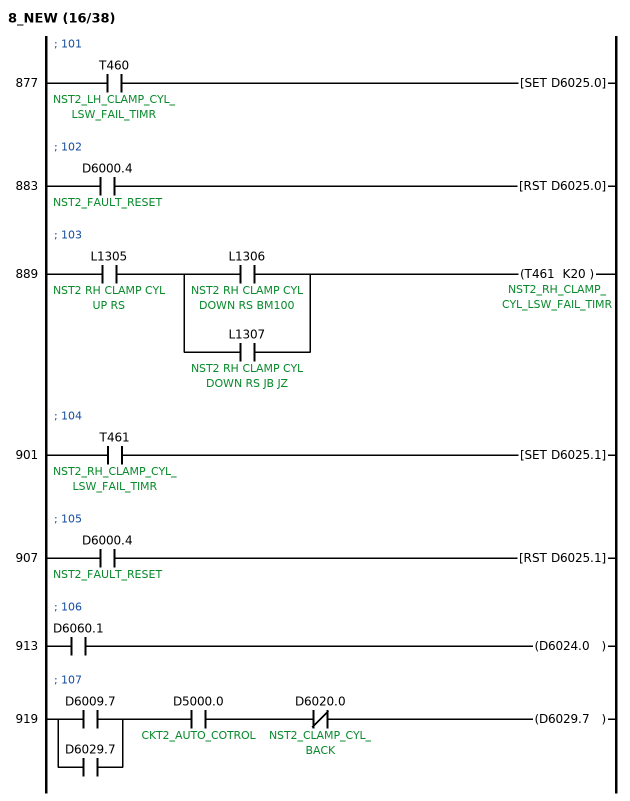
[picture p96: ladder of 8_NEW, rungs at steps 877 to 919]
; 101
877   LD      T460  ; NST2_LH_CLAMP_CYL_LSW_FAIL_TIMR
      SET     D6025.0
; 102
883   LD      D6000.4  ; NST2_FAULT_RESET
      RST     D6025.0
; 103
889   LD      L1305  ; NST2 RH CLAMP CYL UP RS
      LD      L1306  ; NST2 RH CLAMP CYL DOWN RS BM100
      OR      L1307  ; NST2 RH CLAMP CYL DOWN RS JB JZ
      ANB
      OUT     T461 K20  ; NST2_RH_CLAMP_CYL_LSW_FAIL_TIMR
; 104
901   LD      T461  ; NST2_RH_CLAMP_CYL_LSW_FAIL_TIMR
      SET     D6025.1
; 105
907   LD      D6000.4  ; NST2_FAULT_RESET
      RST     D6025.1
; 106
913   LD      D6060.1
      OUT     D6024.0
; 107
919   LD      D6009.7
      OR      D6029.7
      AND     D5000.0  ; CKT2_AUTO_COTROL
      ANI     D6020.0  ; NST2_CLAMP_CYL_BACK
      OUT     D6029.7
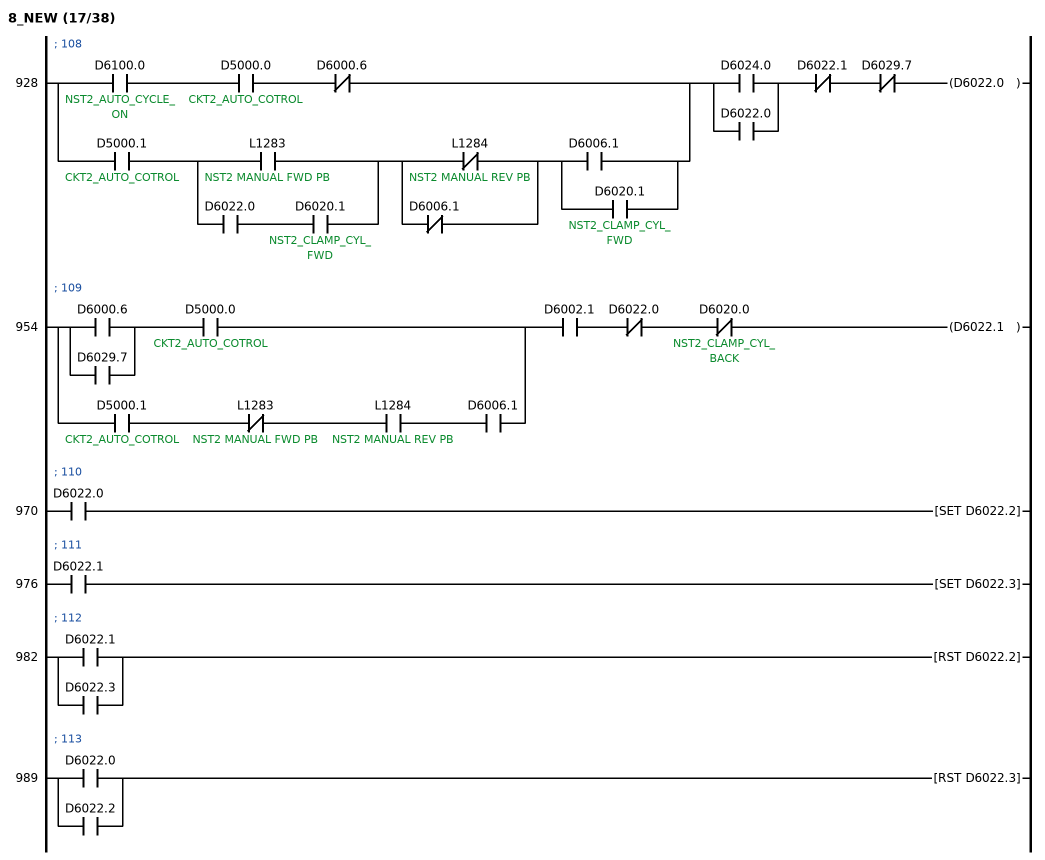
; 108
928   LD      D6100.0  ; NST2_AUTO_CYCLE_ON
      AND     D5000.0  ; CKT2_AUTO_COTROL
      ANI     D6000.6
      LD      D5000.1  ; CKT2_AUTO_COTROL
      LD      L1283  ; NST2 MANUAL FWD PB
      LD      D6022.0
      AND     D6020.1  ; NST2_CLAMP_CYL_FWD
      ORB
      ANB
      LDI     L1284  ; NST2 MANUAL REV PB
      ORI     D6006.1
      ANB
      LD      D6006.1
      OR      D6020.1  ; NST2_CLAMP_CYL_FWD
      ANB
      ORB
      LD      D6024.0
      OR      D6022.0
      ANB
      ANI     D6022.1
      ANI     D6029.7
      OUT     D6022.0
; 109
954   LD      D6000.6
      OR      D6029.7
      AND     D5000.0  ; CKT2_AUTO_COTROL
      LD      D5000.1  ; CKT2_AUTO_COTROL
      ANI     L1283  ; NST2 MANUAL FWD PB
      AND     L1284  ; NST2 MANUAL REV PB
      AND     D6006.1
      ORB
      AND     D6002.1
      ANI     D6022.0
      ANI     D6020.0  ; NST2_CLAMP_CYL_BACK
      OUT     D6022.1
; 110
970   LD      D6022.0
      SET     D6022.2
; 111
976   LD      D6022.1
      SET     D6022.3
; 112
982   LD      D6022.1
      OR      D6022.3
      RST     D6022.2
; 113
989   LD      D6022.0
      OR      D6022.2
      RST     D6022.3
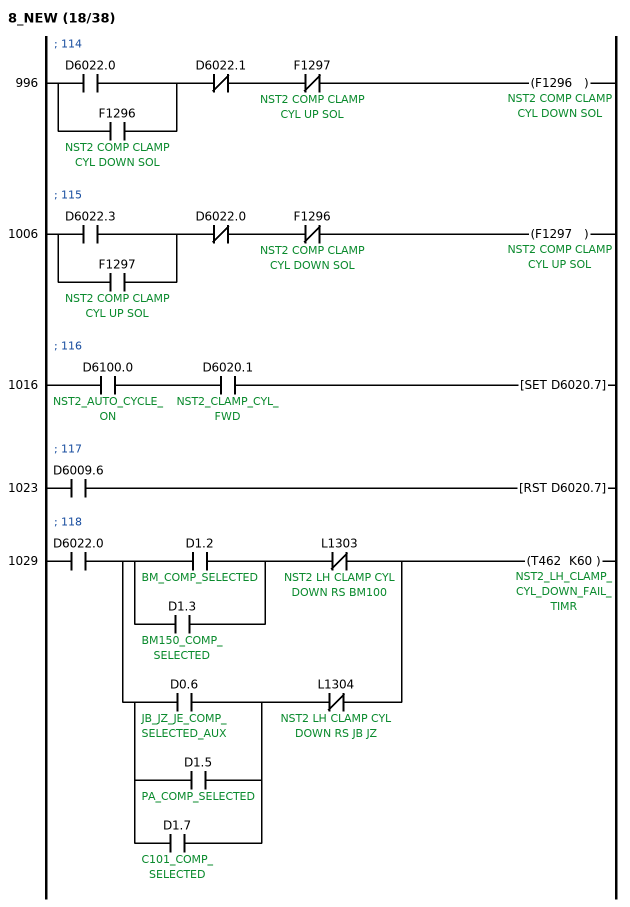
; 114
996   LD      D6022.0
      OR      F1296  ; NST2 COMP CLAMP CYL DOWN SOL
      ANI     D6022.1
      ANI     F1297  ; NST2 COMP CLAMP CYL UP SOL
      OUT     F1296  ; NST2 COMP CLAMP CYL DOWN SOL
; 115
1006  LD      D6022.3
      OR      F1297  ; NST2 COMP CLAMP CYL UP SOL
      ANI     D6022.0
      ANI     F1296  ; NST2 COMP CLAMP CYL DOWN SOL
      OUT     F1297  ; NST2 COMP CLAMP CYL UP SOL
; 116
1016  LD      D6100.0  ; NST2_AUTO_CYCLE_ON
      AND     D6020.1  ; NST2_CLAMP_CYL_FWD
      SET     D6020.7
; 117
1023  LD      D6009.6
      RST     D6020.7
; 118
1029  LD      D6022.0
      LD      D1.2  ; BM_COMP_SELECTED
      OR      D1.3  ; BM150_COMP_SELECTED
      ANI     L1303  ; NST2 LH CLAMP CYL DOWN RS BM100
      LD      D0.6  ; JB_JZ_JE_COMP_SELECTED_AUX
      OR      D1.5  ; PA_COMP_SELECTED
      OR      D1.7  ; C101_COMP_SELECTED
      ANI     L1304  ; NST2 LH CLAMP CYL DOWN RS JB JZ
      ORB
      ANB
      OUT     T462 K60  ; NST2_LH_CLAMP_CYL_DOWN_FAIL_TIMR
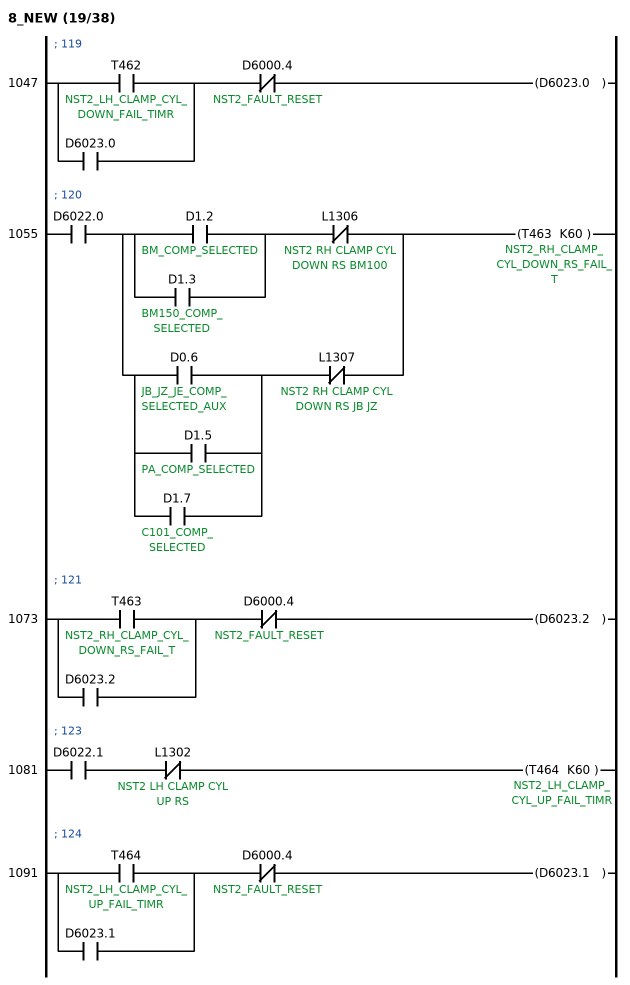
; 119
1047  LD      T462  ; NST2_LH_CLAMP_CYL_DOWN_FAIL_TIMR
      OR      D6023.0
      ANI     D6000.4  ; NST2_FAULT_RESET
      OUT     D6023.0
; 120
1055  LD      D6022.0
      LD      D1.2  ; BM_COMP_SELECTED
      OR      D1.3  ; BM150_COMP_SELECTED
      ANI     L1306  ; NST2 RH CLAMP CYL DOWN RS BM100
      LD      D0.6  ; JB_JZ_JE_COMP_SELECTED_AUX
      OR      D1.5  ; PA_COMP_SELECTED
      OR      D1.7  ; C101_COMP_SELECTED
      ANI     L1307  ; NST2 RH CLAMP CYL DOWN RS JB JZ
      ORB
      ANB
      OUT     T463 K60  ; NST2_RH_CLAMP_CYL_DOWN_RS_FAIL_T
; 121
1073  LD      T463  ; NST2_RH_CLAMP_CYL_DOWN_RS_FAIL_T
      OR      D6023.2
      ANI     D6000.4  ; NST2_FAULT_RESET
      OUT     D6023.2
; 123
1081  LD      D6022.1
      ANI     L1302  ; NST2 LH CLAMP CYL UP RS
      OUT     T464 K60  ; NST2_LH_CLAMP_CYL_UP_FAIL_TIMR
; 124
1091  LD      T464  ; NST2_LH_CLAMP_CYL_UP_FAIL_TIMR
      OR      D6023.1
      ANI     D6000.4  ; NST2_FAULT_RESET
      OUT     D6023.1
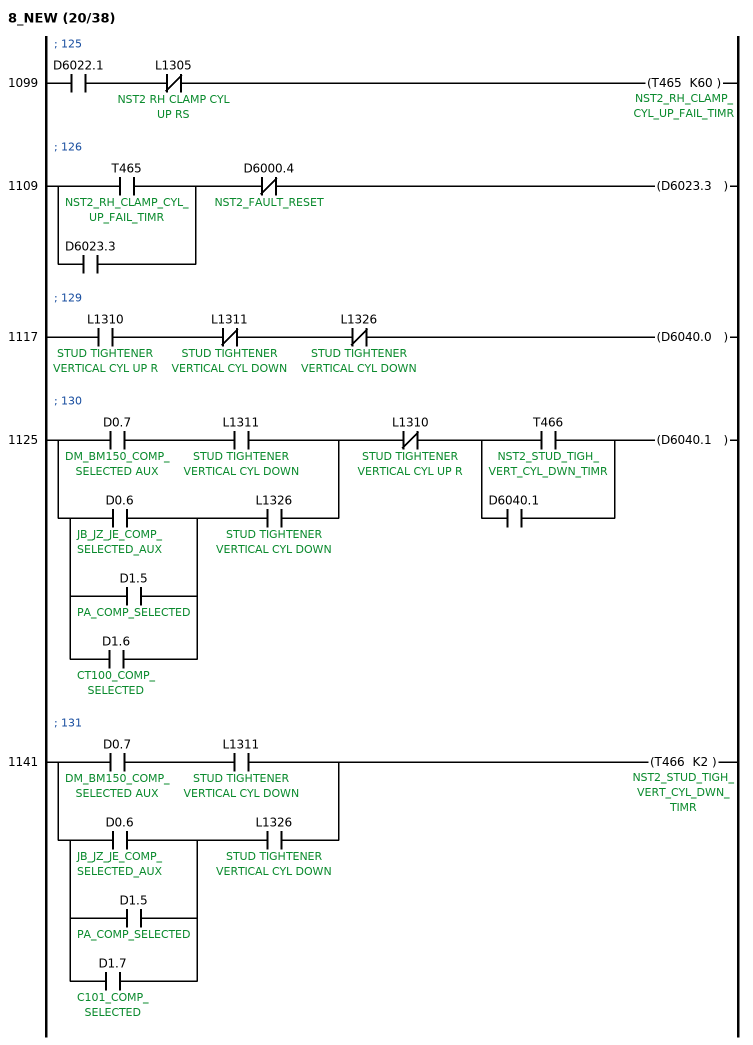
; 125
1099  LD      D6022.1
      ANI     L1305  ; NST2 RH CLAMP CYL UP RS
      OUT     T465 K60  ; NST2_RH_CLAMP_CYL_UP_FAIL_TIMR
; 126
1109  LD      T465  ; NST2_RH_CLAMP_CYL_UP_FAIL_TIMR
      OR      D6023.3
      ANI     D6000.4  ; NST2_FAULT_RESET
      OUT     D6023.3
; 129
1117  LD      L1310  ; STUD TIGHTENER VERTICAL CYL UP R
      ANI     L1311  ; STUD TIGHTENER VERTICAL CYL DOWN
      ANI     L1326  ; STUD TIGHTENER VERTICAL CYL DOWN
      OUT     D6040.0
; 130
1125  LD      D0.7  ; DM_BM150_COMP_SELECTED AUX
      AND     L1311  ; STUD TIGHTENER VERTICAL CYL DOWN
      LD      D0.6  ; JB_JZ_JE_COMP_SELECTED_AUX
      OR      D1.5  ; PA_COMP_SELECTED
      OR      D1.6  ; CT100_COMP_SELECTED
      AND     L1326  ; STUD TIGHTENER VERTICAL CYL DOWN
      ORB
      ANI     L1310  ; STUD TIGHTENER VERTICAL CYL UP R
      LD      T466  ; NST2_STUD_TIGH_VERT_CYL_DWN_TIMR
      OR      D6040.1
      ANB
      OUT     D6040.1
; 131
1141  LD      D0.7  ; DM_BM150_COMP_SELECTED AUX
      AND     L1311  ; STUD TIGHTENER VERTICAL CYL DOWN
      LD      D0.6  ; JB_JZ_JE_COMP_SELECTED_AUX
      OR      D1.5  ; PA_COMP_SELECTED
      OR      D1.7  ; C101_COMP_SELECTED
      AND     L1326  ; STUD TIGHTENER VERTICAL CYL DOWN
      ORB
      OUT     T466 K2  ; NST2_STUD_TIGH_VERT_CYL_DWN_TIMR
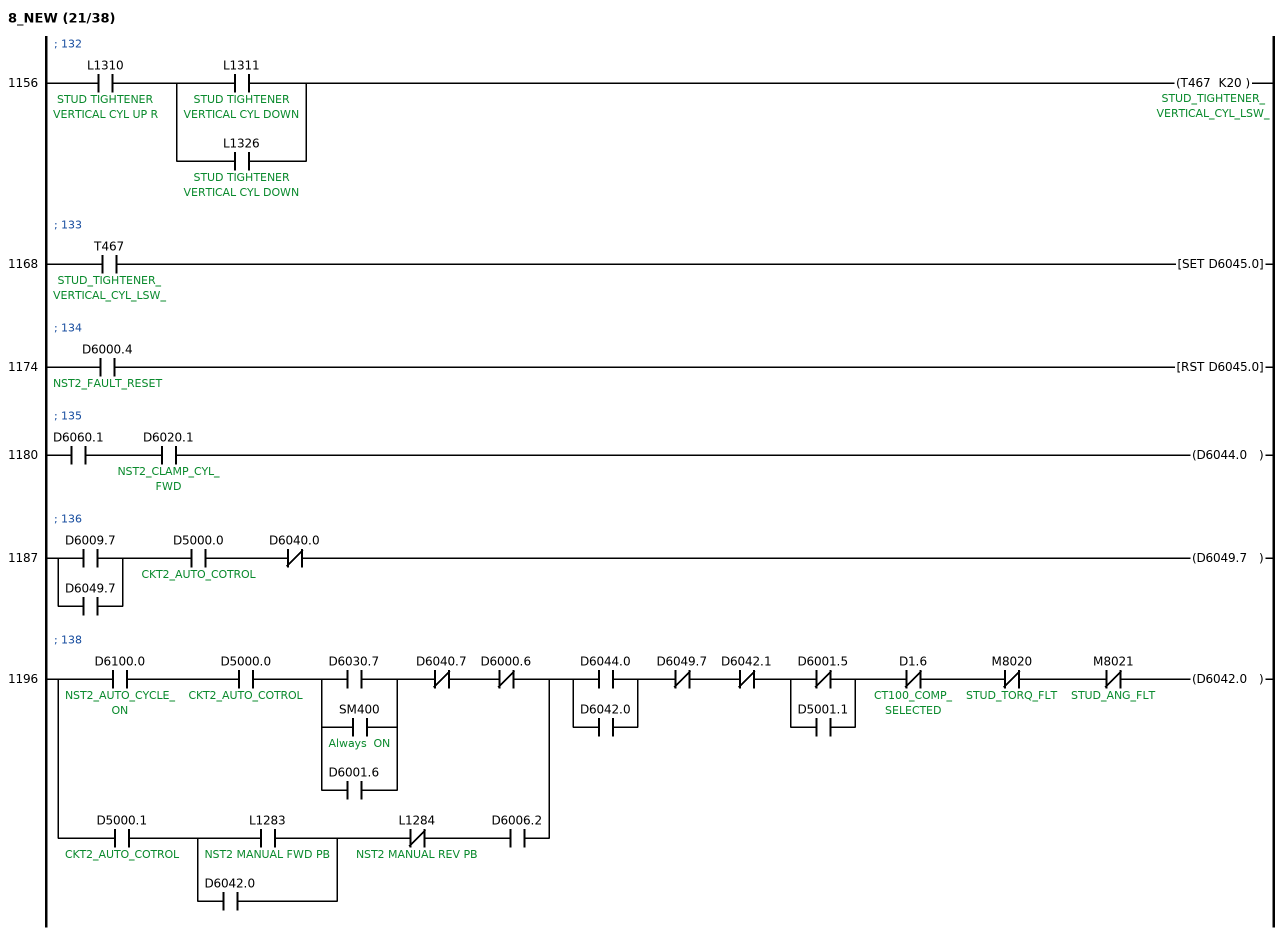
; 132
1156  LD      L1310  ; STUD TIGHTENER VERTICAL CYL UP R
      LD      L1311  ; STUD TIGHTENER VERTICAL CYL DOWN
      OR      L1326  ; STUD TIGHTENER VERTICAL CYL DOWN
      ANB
      OUT     T467 K20  ; STUD_TIGHTENER_VERTICAL_CYL_LSW_
; 133
1168  LD      T467  ; STUD_TIGHTENER_VERTICAL_CYL_LSW_
      SET     D6045.0
; 134
1174  LD      D6000.4  ; NST2_FAULT_RESET
      RST     D6045.0
; 135
1180  LD      D6060.1
      AND     D6020.1  ; NST2_CLAMP_CYL_FWD
      OUT     D6044.0
; 136
1187  LD      D6009.7
      OR      D6049.7
      AND     D5000.0  ; CKT2_AUTO_COTROL
      ANI     D6040.0
      OUT     D6049.7
; 138
1196  LD      D6100.0  ; NST2_AUTO_CYCLE_ON
      AND     D5000.0  ; CKT2_AUTO_COTROL
      LD      D6030.7
      OR      SM400  ; Always  ON
      OR      D6001.6
      ANB
      ANI     D6040.7
      ANI     D6000.6
      LD      D5000.1  ; CKT2_AUTO_COTROL
      LD      L1283  ; NST2 MANUAL FWD PB
      OR      D6042.0
      ANB
      ANI     L1284  ; NST2 MANUAL REV PB
      AND     D6006.2
      ORB
      LD      D6044.0
      OR      D6042.0
      ANB
      ANI     D6049.7
      ANI     D6042.1
      LDI     D6001.5
      OR      D5001.1
      ANB
      ANI     D1.6  ; CT100_COMP_SELECTED
      ANI     M8020  ; STUD_TORQ_FLT
      ANI     M8021  ; STUD_ANG_FLT
      OUT     D6042.0
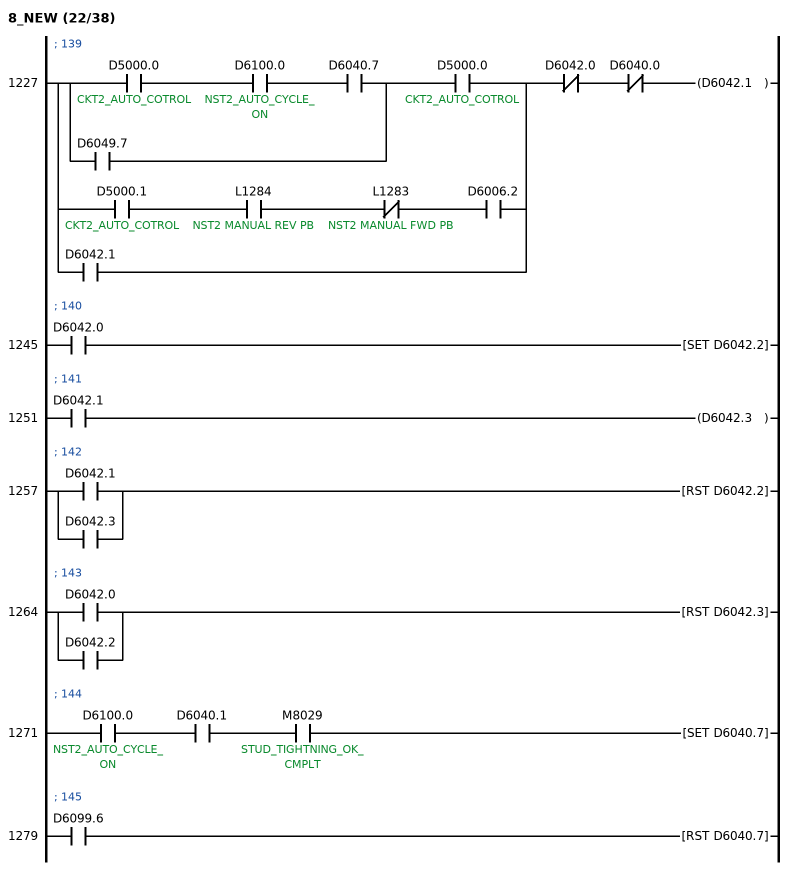
; 139
1227  LD      D5000.0  ; CKT2_AUTO_COTROL
      AND     D6100.0  ; NST2_AUTO_CYCLE_ON
      AND     D6040.7
      OR      D6049.7
      AND     D5000.0  ; CKT2_AUTO_COTROL
      LD      D5000.1  ; CKT2_AUTO_COTROL
      AND     L1284  ; NST2 MANUAL REV PB
      ANI     L1283  ; NST2 MANUAL FWD PB
      AND     D6006.2
      ORB
      OR      D6042.1
      ANI     D6042.0
      ANI     D6040.0
      OUT     D6042.1
; 140
1245  LD      D6042.0
      SET     D6042.2
; 141
1251  LD      D6042.1
      OUT     D6042.3
; 142
1257  LD      D6042.1
      OR      D6042.3
      RST     D6042.2
; 143
1264  LD      D6042.0
      OR      D6042.2
      RST     D6042.3
; 144
1271  LD      D6100.0  ; NST2_AUTO_CYCLE_ON
      AND     D6040.1
      AND     M8029  ; STUD_TIGHTNING_OK_CMPLT
      SET     D6040.7
; 145
1279  LD      D6099.6
      RST     D6040.7
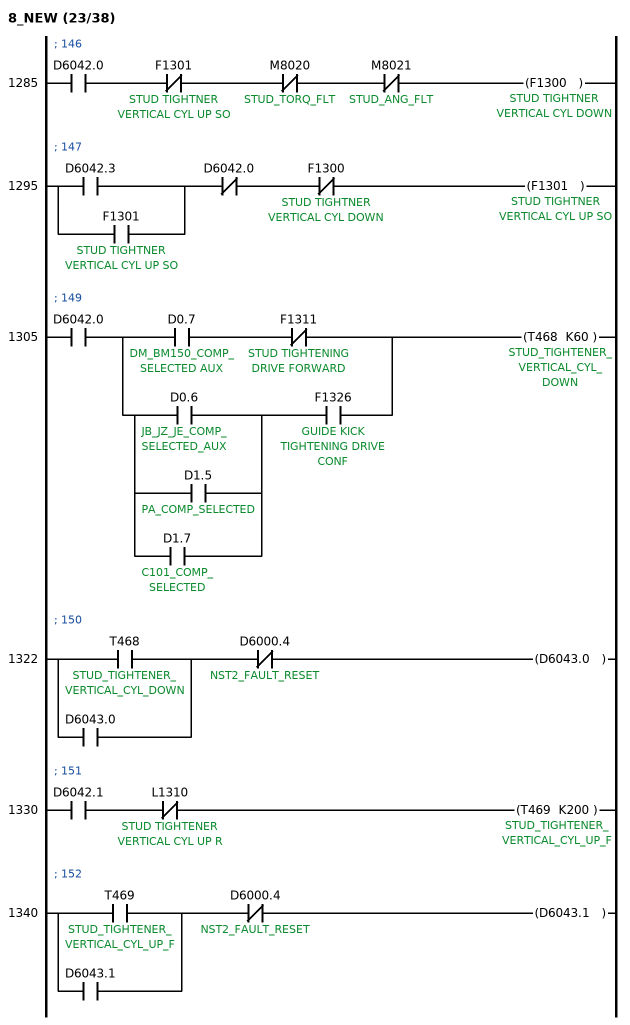
; 146
1285  LD      D6042.0
      ANI     F1301  ; STUD TIGHTNER VERTICAL CYL UP SO
      ANI     M8020  ; STUD_TORQ_FLT
      ANI     M8021  ; STUD_ANG_FLT
      OUT     F1300  ; STUD TIGHTNER VERTICAL CYL DOWN
; 147
1295  LD      D6042.3
      OR      F1301  ; STUD TIGHTNER VERTICAL CYL UP SO
      ANI     D6042.0
      ANI     F1300  ; STUD TIGHTNER VERTICAL CYL DOWN
      OUT     F1301  ; STUD TIGHTNER VERTICAL CYL UP SO
; 149
1305  LD      D6042.0
      LD      D0.7  ; DM_BM150_COMP_SELECTED AUX
      ANI     F1311  ; STUD TIGHTENING DRIVE FORWARD
      LD      D0.6  ; JB_JZ_JE_COMP_SELECTED_AUX
      OR      D1.5  ; PA_COMP_SELECTED
      OR      D1.7  ; C101_COMP_SELECTED
      AND     F1326  ; GUIDE KICK TIGHTENING DRIVE CONF
      ORB
      ANB
      OUT     T468 K60  ; STUD_TIGHTENER_VERTICAL_CYL_DOWN
; 150
1322  LD      T468  ; STUD_TIGHTENER_VERTICAL_CYL_DOWN
      OR      D6043.0
      ANI     D6000.4  ; NST2_FAULT_RESET
      OUT     D6043.0
; 151
1330  LD      D6042.1
      ANI     L1310  ; STUD TIGHTENER VERTICAL CYL UP R
      OUT     T469 K200  ; STUD_TIGHTENER_VERTICAL_CYL_UP_F
; 152
1340  LD      T469  ; STUD_TIGHTENER_VERTICAL_CYL_UP_F
      OR      D6043.1
      ANI     D6000.4  ; NST2_FAULT_RESET
      OUT     D6043.1
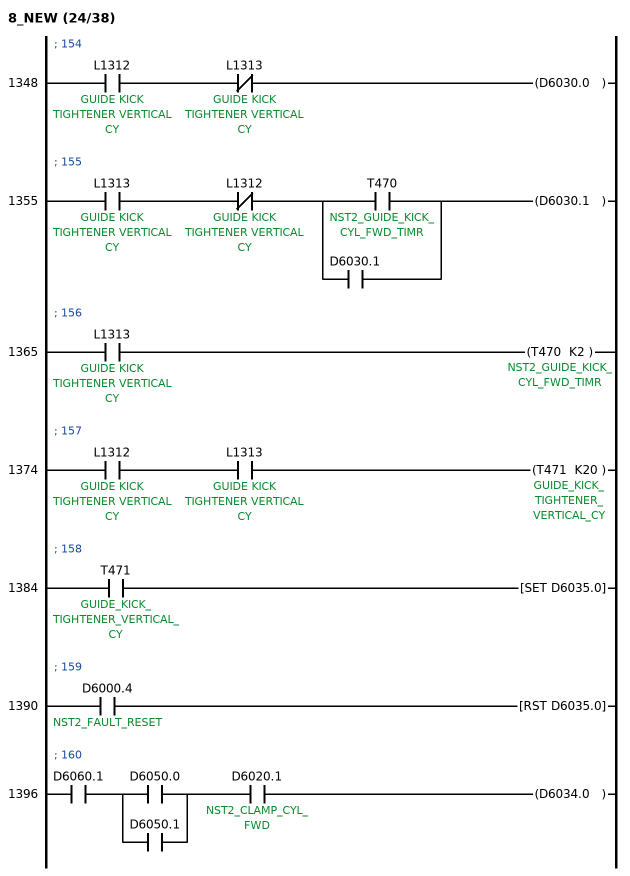
; 154
1348  LD      L1312  ; GUIDE KICK TIGHTENER VERTICAL CY
      ANI     L1313  ; GUIDE KICK TIGHTENER VERTICAL CY
      OUT     D6030.0
; 155
1355  LD      L1313  ; GUIDE KICK TIGHTENER VERTICAL CY
      ANI     L1312  ; GUIDE KICK TIGHTENER VERTICAL CY
      LD      T470  ; NST2_GUIDE_KICK_CYL_FWD_TIMR
      OR      D6030.1
      ANB
      OUT     D6030.1
; 156
1365  LD      L1313  ; GUIDE KICK TIGHTENER VERTICAL CY
      OUT     T470 K2  ; NST2_GUIDE_KICK_CYL_FWD_TIMR
; 157
1374  LD      L1312  ; GUIDE KICK TIGHTENER VERTICAL CY
      AND     L1313  ; GUIDE KICK TIGHTENER VERTICAL CY
      OUT     T471 K20  ; GUIDE_KICK_TIGHTENER_VERTICAL_CY
; 158
1384  LD      T471  ; GUIDE_KICK_TIGHTENER_VERTICAL_CY
      SET     D6035.0
; 159
1390  LD      D6000.4  ; NST2_FAULT_RESET
      RST     D6035.0
; 160
1396  LD      D6060.1
      LD      D6050.0
      OR      D6050.1
      ANB
      AND     D6020.1  ; NST2_CLAMP_CYL_FWD
      OUT     D6034.0
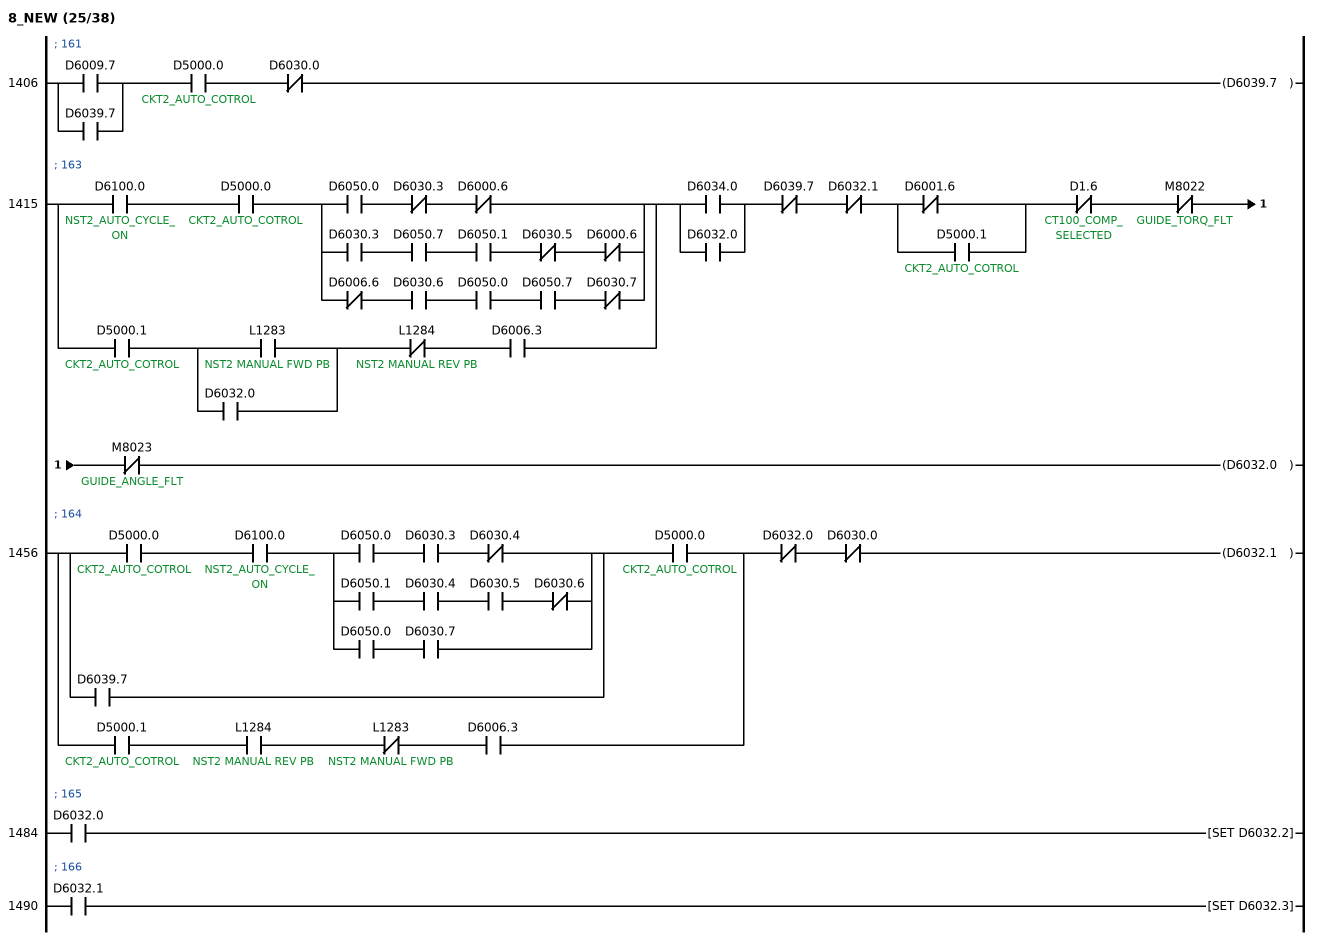
; 161
1406  LD      D6009.7
      OR      D6039.7
      AND     D5000.0  ; CKT2_AUTO_COTROL
      ANI     D6030.0
      OUT     D6039.7
; 163
1415  LD      D6100.0  ; NST2_AUTO_CYCLE_ON
      AND     D5000.0  ; CKT2_AUTO_COTROL
      LD      D6050.0
      ANI     D6030.3
      ANI     D6000.6
      LD      D6030.3
      AND     D6050.7
      AND     D6050.1
      ANI     D6030.5
      ANI     D6000.6
      ORB
      LDI     D6006.6
      AND     D6030.6
      AND     D6050.0
      AND     D6050.7
      ANI     D6030.7
      ORB
      ANB
      LD      D5000.1  ; CKT2_AUTO_COTROL
      LD      L1283  ; NST2 MANUAL FWD PB
      OR      D6032.0
      ANB
      ANI     L1284  ; NST2 MANUAL REV PB
      AND     D6006.3
      ORB
      LD      D6034.0
      OR      D6032.0
      ANB
      ANI     D6039.7
      ANI     D6032.1
      LDI     D6001.6
      OR      D5000.1  ; CKT2_AUTO_COTROL
      ANB
      ANI     D1.6  ; CT100_COMP_SELECTED
      ANI     M8022  ; GUIDE_TORQ_FLT
      ANI     M8023  ; GUIDE_ANGLE_FLT
      OUT     D6032.0
; 164
1456  LD      D5000.0  ; CKT2_AUTO_COTROL
      AND     D6100.0  ; NST2_AUTO_CYCLE_ON
      LD      D6050.0
      AND     D6030.3
      ANI     D6030.4
      LD      D6050.1
      AND     D6030.4
      AND     D6030.5
      ANI     D6030.6
      ORB
      LD      D6050.0
      AND     D6030.7
      ORB
      ANB
      OR      D6039.7
      AND     D5000.0  ; CKT2_AUTO_COTROL
      LD      D5000.1  ; CKT2_AUTO_COTROL
      AND     L1284  ; NST2 MANUAL REV PB
      ANI     L1283  ; NST2 MANUAL FWD PB
      AND     D6006.3
      ORB
      ANI     D6032.0
      ANI     D6030.0
      OUT     D6032.1
; 165
1484  LD      D6032.0
      SET     D6032.2
; 166
1490  LD      D6032.1
      SET     D6032.3
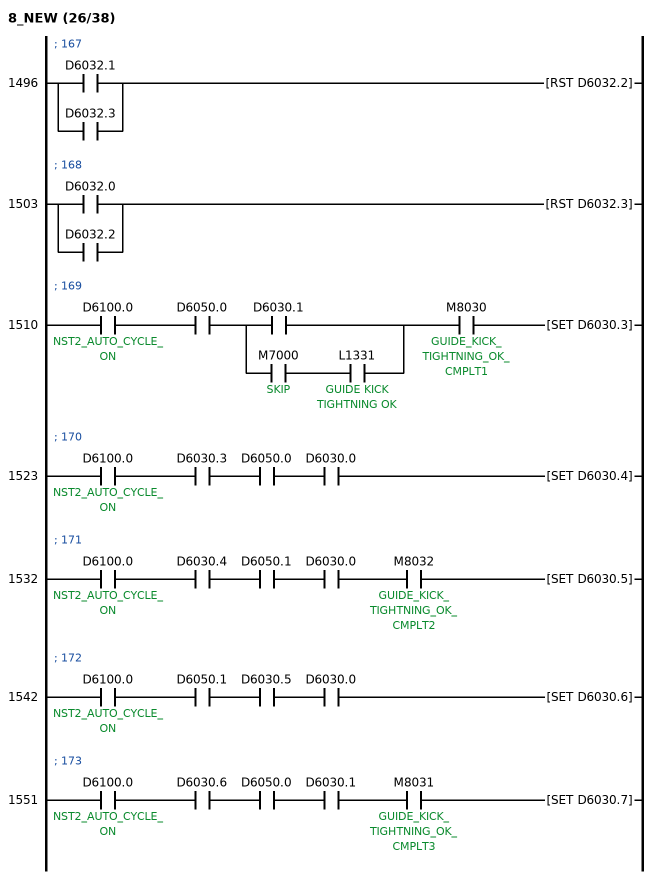
; 167
1496  LD      D6032.1
      OR      D6032.3
      RST     D6032.2
; 168
1503  LD      D6032.0
      OR      D6032.2
      RST     D6032.3
; 169
1510  LD      D6100.0  ; NST2_AUTO_CYCLE_ON
      AND     D6050.0
      LD      D6030.1
      LD      M7000  ; SKIP
      AND     L1331  ; GUIDE KICK TIGHTNING OK
      ORB
      ANB
      AND     M8030  ; GUIDE_KICK_TIGHTNING_OK_CMPLT1
      SET     D6030.3
; 170
1523  LD      D6100.0  ; NST2_AUTO_CYCLE_ON
      AND     D6030.3
      AND     D6050.0
      AND     D6030.0
      SET     D6030.4
; 171
1532  LD      D6100.0  ; NST2_AUTO_CYCLE_ON
      AND     D6030.4
      AND     D6050.1
      AND     D6030.0
      AND     M8032  ; GUIDE_KICK_TIGHTNING_OK_CMPLT2
      SET     D6030.5
; 172
1542  LD      D6100.0  ; NST2_AUTO_CYCLE_ON
      AND     D6050.1
      AND     D6030.5
      AND     D6030.0
      SET     D6030.6
; 173
1551  LD      D6100.0  ; NST2_AUTO_CYCLE_ON
      AND     D6030.6
      AND     D6050.0
      AND     D6030.1
      AND     M8031  ; GUIDE_KICK_TIGHTNING_OK_CMPLT3
      SET     D6030.7
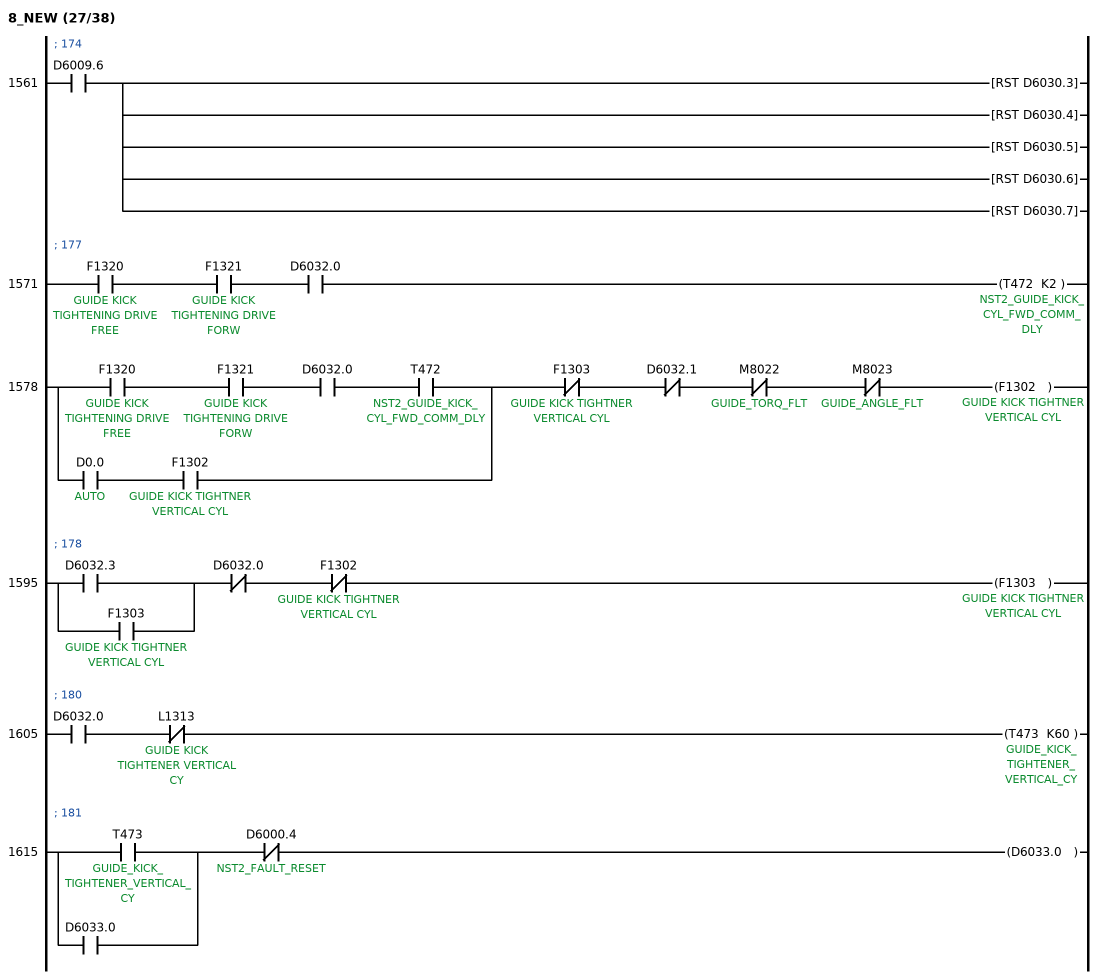
; 174
1561  LD      D6009.6
      RST     D6030.3
      RST     D6030.4
      RST     D6030.5
      RST     D6030.6
      RST     D6030.7
; 177
1571  LD      F1320  ; GUIDE KICK TIGHTENING DRIVE FREE
      AND     F1321  ; GUIDE KICK TIGHTENING DRIVE FORW
      AND     D6032.0
      OUT     T472 K2  ; NST2_GUIDE_KICK_CYL_FWD_COMM_DLY
1578  LD      F1320  ; GUIDE KICK TIGHTENING DRIVE FREE
      AND     F1321  ; GUIDE KICK TIGHTENING DRIVE FORW
      AND     D6032.0
      AND     T472  ; NST2_GUIDE_KICK_CYL_FWD_COMM_DLY
      LD      D0.0  ; AUTO
      AND     F1302  ; GUIDE KICK TIGHTNER VERTICAL CYL
      ORB
      ANI     F1303  ; GUIDE KICK TIGHTNER VERTICAL CYL
      ANI     D6032.1
      ANI     M8022  ; GUIDE_TORQ_FLT
      ANI     M8023  ; GUIDE_ANGLE_FLT
      OUT     F1302  ; GUIDE KICK TIGHTNER VERTICAL CYL
; 178
1595  LD      D6032.3
      OR      F1303  ; GUIDE KICK TIGHTNER VERTICAL CYL
      ANI     D6032.0
      ANI     F1302  ; GUIDE KICK TIGHTNER VERTICAL CYL
      OUT     F1303  ; GUIDE KICK TIGHTNER VERTICAL CYL
; 180
1605  LD      D6032.0
      ANI     L1313  ; GUIDE KICK TIGHTENER VERTICAL CY
      OUT     T473 K60  ; GUIDE_KICK_TIGHTENER_VERTICAL_CY
; 181
1615  LD      T473  ; GUIDE_KICK_TIGHTENER_VERTICAL_CY
      OR      D6033.0
      ANI     D6000.4  ; NST2_FAULT_RESET
      OUT     D6033.0
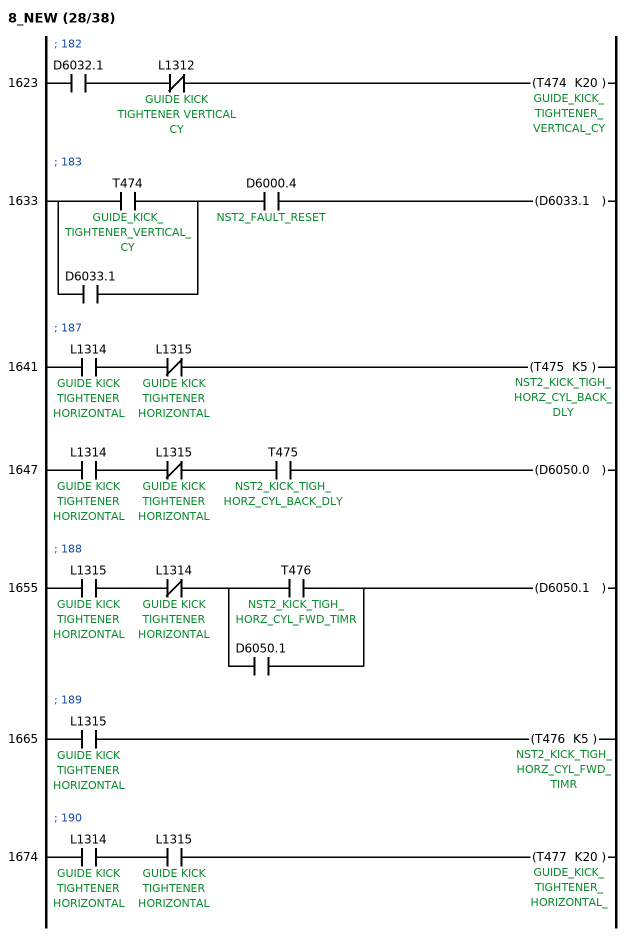
; 182
1623  LD      D6032.1
      ANI     L1312  ; GUIDE KICK TIGHTENER VERTICAL CY
      OUT     T474 K20  ; GUIDE_KICK_TIGHTENER_VERTICAL_CY
; 183
1633  LD      T474  ; GUIDE_KICK_TIGHTENER_VERTICAL_CY
      OR      D6033.1
      AND     D6000.4  ; NST2_FAULT_RESET
      OUT     D6033.1
; 187
1641  LD      L1314  ; GUIDE KICK TIGHTENER HORIZONTAL
      ANI     L1315  ; GUIDE KICK TIGHTENER HORIZONTAL
      OUT     T475 K5  ; NST2_KICK_TIGH_HORZ_CYL_BACK_DLY
1647  LD      L1314  ; GUIDE KICK TIGHTENER HORIZONTAL
      ANI     L1315  ; GUIDE KICK TIGHTENER HORIZONTAL
      AND     T475  ; NST2_KICK_TIGH_HORZ_CYL_BACK_DLY
      OUT     D6050.0
; 188
1655  LD      L1315  ; GUIDE KICK TIGHTENER HORIZONTAL
      ANI     L1314  ; GUIDE KICK TIGHTENER HORIZONTAL
      LD      T476  ; NST2_KICK_TIGH_HORZ_CYL_FWD_TIMR
      OR      D6050.1
      ANB
      OUT     D6050.1
; 189
1665  LD      L1315  ; GUIDE KICK TIGHTENER HORIZONTAL
      OUT     T476 K5  ; NST2_KICK_TIGH_HORZ_CYL_FWD_TIMR
; 190
1674  LD      L1314  ; GUIDE KICK TIGHTENER HORIZONTAL
      AND     L1315  ; GUIDE KICK TIGHTENER HORIZONTAL
      OUT     T477 K20  ; GUIDE_KICK_TIGHTENER_HORIZONTAL_
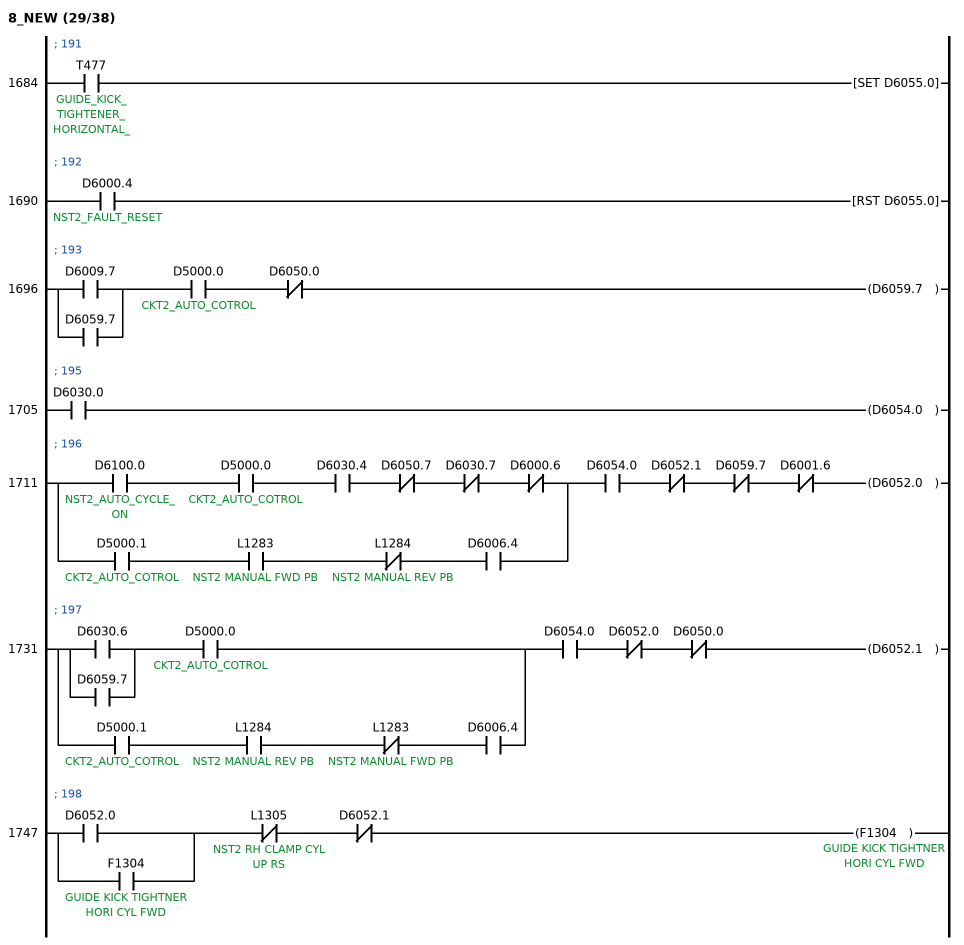
; 191
1684  LD      T477  ; GUIDE_KICK_TIGHTENER_HORIZONTAL_
      SET     D6055.0
; 192
1690  LD      D6000.4  ; NST2_FAULT_RESET
      RST     D6055.0
; 193
1696  LD      D6009.7
      OR      D6059.7
      AND     D5000.0  ; CKT2_AUTO_COTROL
      ANI     D6050.0
      OUT     D6059.7
; 195
1705  LD      D6030.0
      OUT     D6054.0
; 196
1711  LD      D6100.0  ; NST2_AUTO_CYCLE_ON
      AND     D5000.0  ; CKT2_AUTO_COTROL
      AND     D6030.4
      ANI     D6050.7
      ANI     D6030.7
      ANI     D6000.6
      LD      D5000.1  ; CKT2_AUTO_COTROL
      AND     L1283  ; NST2 MANUAL FWD PB
      ANI     L1284  ; NST2 MANUAL REV PB
      AND     D6006.4
      ORB
      AND     D6054.0
      ANI     D6052.1
      ANI     D6059.7
      ANI     D6001.6
      OUT     D6052.0
; 197
1731  LD      D6030.6
      OR      D6059.7
      AND     D5000.0  ; CKT2_AUTO_COTROL
      LD      D5000.1  ; CKT2_AUTO_COTROL
      AND     L1284  ; NST2 MANUAL REV PB
      ANI     L1283  ; NST2 MANUAL FWD PB
      AND     D6006.4
      ORB
      AND     D6054.0
      ANI     D6052.0
      ANI     D6050.0
      OUT     D6052.1
; 198
1747  LD      D6052.0
      OR      F1304  ; GUIDE KICK TIGHTNER HORI CYL FWD
      ANI     L1305  ; NST2 RH CLAMP CYL UP RS
      ANI     D6052.1
      OUT     F1304  ; GUIDE KICK TIGHTNER HORI CYL FWD
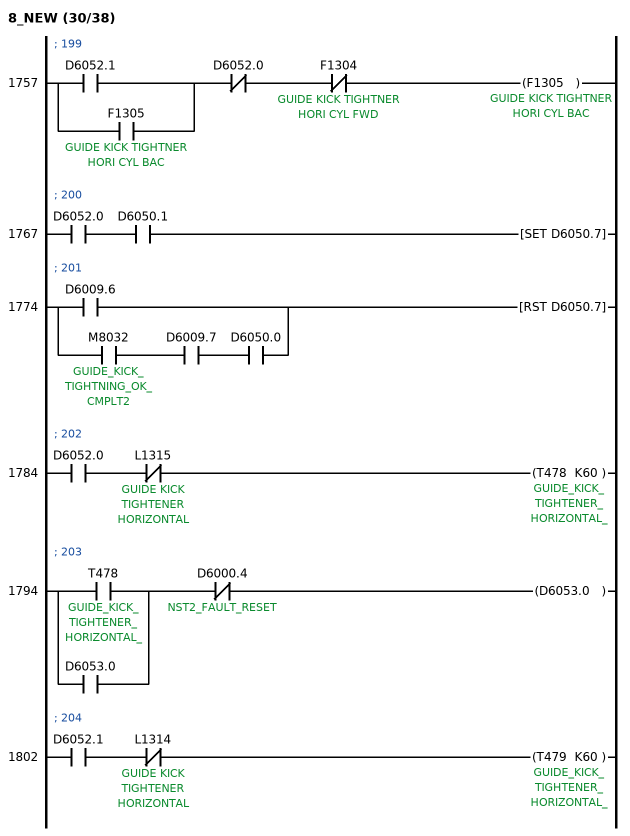
; 199
1757  LD      D6052.1
      OR      F1305  ; GUIDE KICK TIGHTNER HORI CYL BAC
      ANI     D6052.0
      ANI     F1304  ; GUIDE KICK TIGHTNER HORI CYL FWD
      OUT     F1305  ; GUIDE KICK TIGHTNER HORI CYL BAC
; 200
1767  LD      D6052.0
      AND     D6050.1
      SET     D6050.7
; 201
1774  LD      D6009.6
      LD      M8032  ; GUIDE_KICK_TIGHTNING_OK_CMPLT2
      AND     D6009.7
      AND     D6050.0
      ORB
      RST     D6050.7
; 202
1784  LD      D6052.0
      ANI     L1315  ; GUIDE KICK TIGHTENER HORIZONTAL
      OUT     T478 K60  ; GUIDE_KICK_TIGHTENER_HORIZONTAL_
; 203
1794  LD      T478  ; GUIDE_KICK_TIGHTENER_HORIZONTAL_
      OR      D6053.0
      ANI     D6000.4  ; NST2_FAULT_RESET
      OUT     D6053.0
; 204
1802  LD      D6052.1
      ANI     L1314  ; GUIDE KICK TIGHTENER HORIZONTAL
      OUT     T479 K60  ; GUIDE_KICK_TIGHTENER_HORIZONTAL_
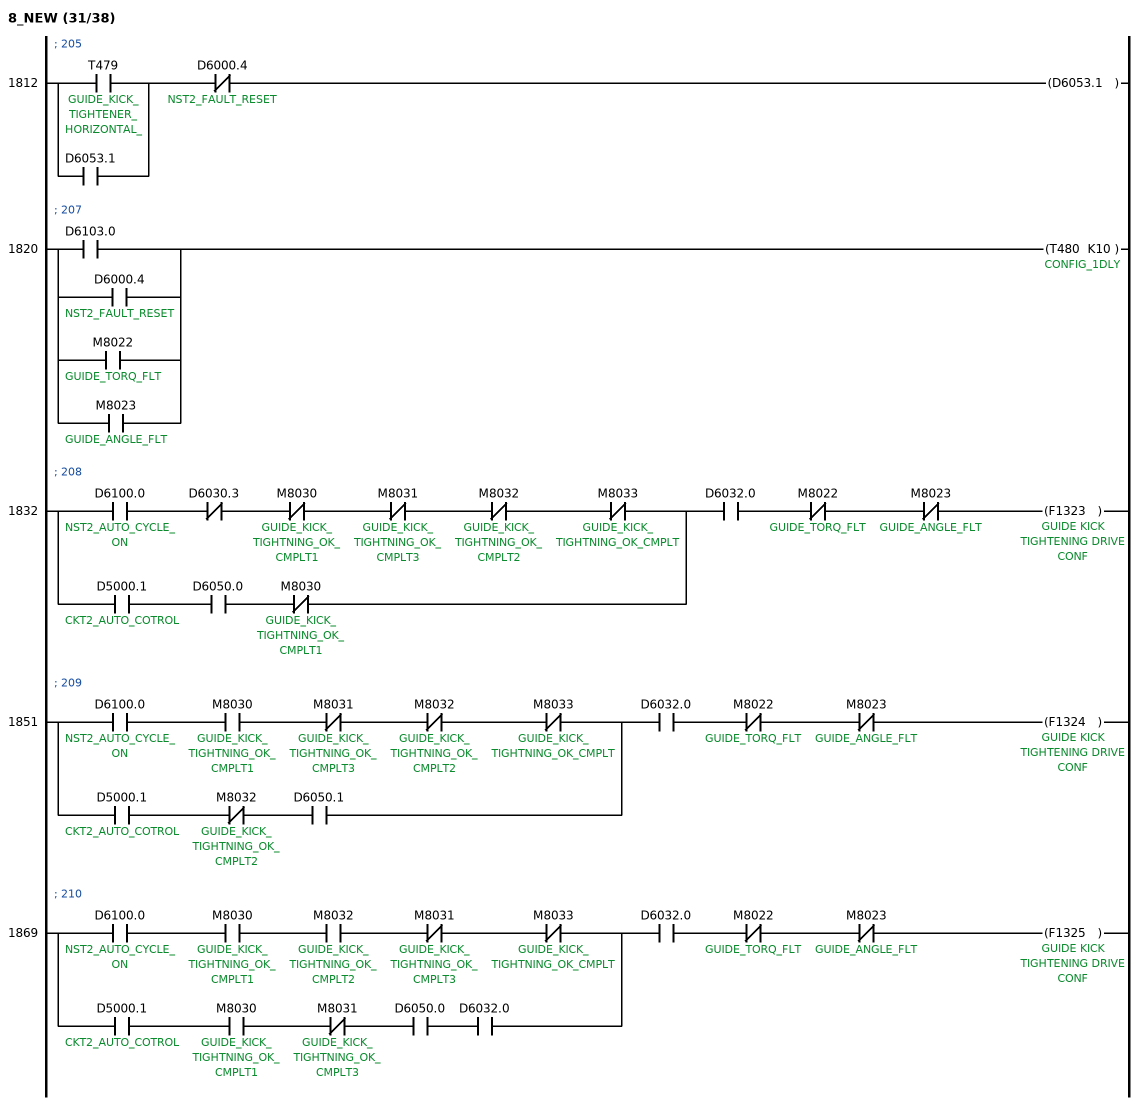
; 205
1812  LD      T479  ; GUIDE_KICK_TIGHTENER_HORIZONTAL_
      OR      D6053.1
      ANI     D6000.4  ; NST2_FAULT_RESET
      OUT     D6053.1
; 207
1820  LD      D6103.0
      OR      D6000.4  ; NST2_FAULT_RESET
      OR      M8022  ; GUIDE_TORQ_FLT
      OR      M8023  ; GUIDE_ANGLE_FLT
      OUT     T480 K10  ; CONFIG_1DLY
; 208
1832  LD      D6100.0  ; NST2_AUTO_CYCLE_ON
      ANI     D6030.3
      ANI     M8030  ; GUIDE_KICK_TIGHTNING_OK_CMPLT1
      ANI     M8031  ; GUIDE_KICK_TIGHTNING_OK_CMPLT3
      ANI     M8032  ; GUIDE_KICK_TIGHTNING_OK_CMPLT2
      ANI     M8033  ; GUIDE_KICK_TIGHTNING_OK_CMPLT
      LD      D5000.1  ; CKT2_AUTO_COTROL
      AND     D6050.0
      ANI     M8030  ; GUIDE_KICK_TIGHTNING_OK_CMPLT1
      ORB
      AND     D6032.0
      ANI     M8022  ; GUIDE_TORQ_FLT
      ANI     M8023  ; GUIDE_ANGLE_FLT
      OUT     F1323  ; GUIDE KICK TIGHTENING DRIVE CONF
; 209
1851  LD      D6100.0  ; NST2_AUTO_CYCLE_ON
      AND     M8030  ; GUIDE_KICK_TIGHTNING_OK_CMPLT1
      ANI     M8031  ; GUIDE_KICK_TIGHTNING_OK_CMPLT3
      ANI     M8032  ; GUIDE_KICK_TIGHTNING_OK_CMPLT2
      ANI     M8033  ; GUIDE_KICK_TIGHTNING_OK_CMPLT
      LD      D5000.1  ; CKT2_AUTO_COTROL
      ANI     M8032  ; GUIDE_KICK_TIGHTNING_OK_CMPLT2
      AND     D6050.1
      ORB
      AND     D6032.0
      ANI     M8022  ; GUIDE_TORQ_FLT
      ANI     M8023  ; GUIDE_ANGLE_FLT
      OUT     F1324  ; GUIDE KICK TIGHTENING DRIVE CONF
; 210
1869  LD      D6100.0  ; NST2_AUTO_CYCLE_ON
      AND     M8030  ; GUIDE_KICK_TIGHTNING_OK_CMPLT1
      AND     M8032  ; GUIDE_KICK_TIGHTNING_OK_CMPLT2
      ANI     M8031  ; GUIDE_KICK_TIGHTNING_OK_CMPLT3
      ANI     M8033  ; GUIDE_KICK_TIGHTNING_OK_CMPLT
      LD      D5000.1  ; CKT2_AUTO_COTROL
      AND     M8030  ; GUIDE_KICK_TIGHTNING_OK_CMPLT1
      ANI     M8031  ; GUIDE_KICK_TIGHTNING_OK_CMPLT3
      AND     D6050.0
      AND     D6032.0
      ORB
      AND     D6032.0
      ANI     M8022  ; GUIDE_TORQ_FLT
      ANI     M8023  ; GUIDE_ANGLE_FLT
      OUT     F1325  ; GUIDE KICK TIGHTENING DRIVE CONF
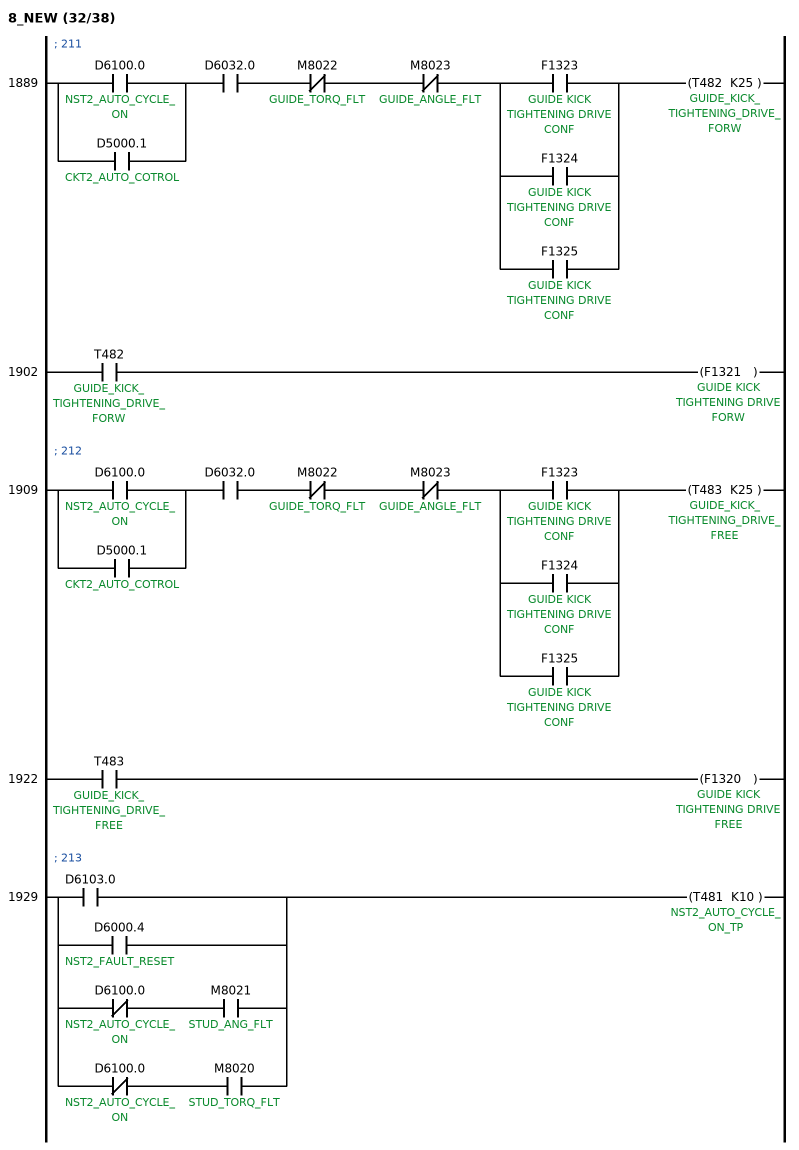
; 211
1889  LD      D6100.0  ; NST2_AUTO_CYCLE_ON
      OR      D5000.1  ; CKT2_AUTO_COTROL
      AND     D6032.0
      ANI     M8022  ; GUIDE_TORQ_FLT
      ANI     M8023  ; GUIDE_ANGLE_FLT
      LD      F1323  ; GUIDE KICK TIGHTENING DRIVE CONF
      OR      F1324  ; GUIDE KICK TIGHTENING DRIVE CONF
      OR      F1325  ; GUIDE KICK TIGHTENING DRIVE CONF
      ANB
      OUT     T482 K25  ; GUIDE_KICK_TIGHTENING_DRIVE_FORW
1902  LD      T482  ; GUIDE_KICK_TIGHTENING_DRIVE_FORW
      OUT     F1321  ; GUIDE KICK TIGHTENING DRIVE FORW
; 212
1909  LD      D6100.0  ; NST2_AUTO_CYCLE_ON
      OR      D5000.1  ; CKT2_AUTO_COTROL
      AND     D6032.0
      ANI     M8022  ; GUIDE_TORQ_FLT
      ANI     M8023  ; GUIDE_ANGLE_FLT
      LD      F1323  ; GUIDE KICK TIGHTENING DRIVE CONF
      OR      F1324  ; GUIDE KICK TIGHTENING DRIVE CONF
      OR      F1325  ; GUIDE KICK TIGHTENING DRIVE CONF
      ANB
      OUT     T483 K25  ; GUIDE_KICK_TIGHTENING_DRIVE_FREE
1922  LD      T483  ; GUIDE_KICK_TIGHTENING_DRIVE_FREE
      OUT     F1320  ; GUIDE KICK TIGHTENING DRIVE FREE
; 213
1929  LD      D6103.0
      OR      D6000.4  ; NST2_FAULT_RESET
      LDI     D6100.0  ; NST2_AUTO_CYCLE_ON
      AND     M8021  ; STUD_ANG_FLT
      ORB
      LDI     D6100.0  ; NST2_AUTO_CYCLE_ON
      AND     M8020  ; STUD_TORQ_FLT
      ORB
      OUT     T481 K10  ; NST2_AUTO_CYCLE_ON_TP
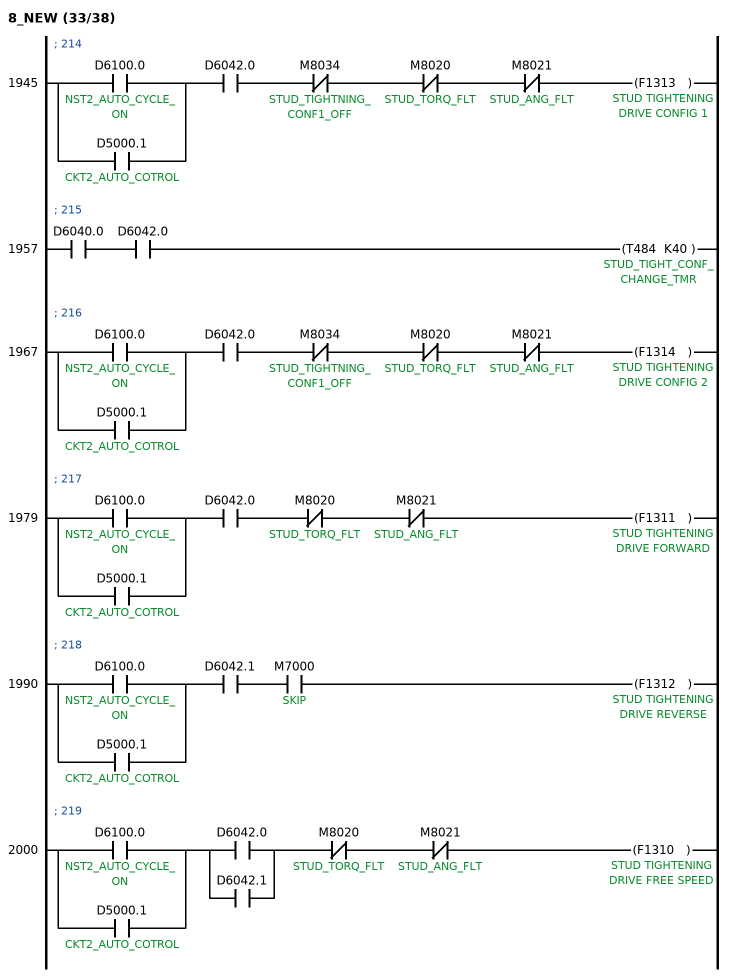
; 214
1945  LD      D6100.0  ; NST2_AUTO_CYCLE_ON
      OR      D5000.1  ; CKT2_AUTO_COTROL
      AND     D6042.0
      ANI     M8034  ; STUD_TIGHTNING_CONF1_OFF
      ANI     M8020  ; STUD_TORQ_FLT
      ANI     M8021  ; STUD_ANG_FLT
      OUT     F1313  ; STUD TIGHTENING DRIVE CONFIG 1
; 215
1957  LD      D6040.0
      AND     D6042.0
      OUT     T484 K40  ; STUD_TIGHT_CONF_CHANGE_TMR
; 216
1967  LD      D6100.0  ; NST2_AUTO_CYCLE_ON
      OR      D5000.1  ; CKT2_AUTO_COTROL
      AND     D6042.0
      ANI     M8034  ; STUD_TIGHTNING_CONF1_OFF
      ANI     M8020  ; STUD_TORQ_FLT
      ANI     M8021  ; STUD_ANG_FLT
      OUT     F1314  ; STUD TIGHTENING DRIVE CONFIG 2
; 217
1979  LD      D6100.0  ; NST2_AUTO_CYCLE_ON
      OR      D5000.1  ; CKT2_AUTO_COTROL
      AND     D6042.0
      ANI     M8020  ; STUD_TORQ_FLT
      ANI     M8021  ; STUD_ANG_FLT
      OUT     F1311  ; STUD TIGHTENING DRIVE FORWARD
; 218
1990  LD      D6100.0  ; NST2_AUTO_CYCLE_ON
      OR      D5000.1  ; CKT2_AUTO_COTROL
      AND     D6042.1
      AND     M7000  ; SKIP
      OUT     F1312  ; STUD TIGHTENING DRIVE REVERSE
; 219
2000  LD      D6100.0  ; NST2_AUTO_CYCLE_ON
      OR      D5000.1  ; CKT2_AUTO_COTROL
      LD      D6042.0
      OR      D6042.1
      ANB
      ANI     M8020  ; STUD_TORQ_FLT
      ANI     M8021  ; STUD_ANG_FLT
      OUT     F1310  ; STUD TIGHTENING DRIVE FREE SPEED
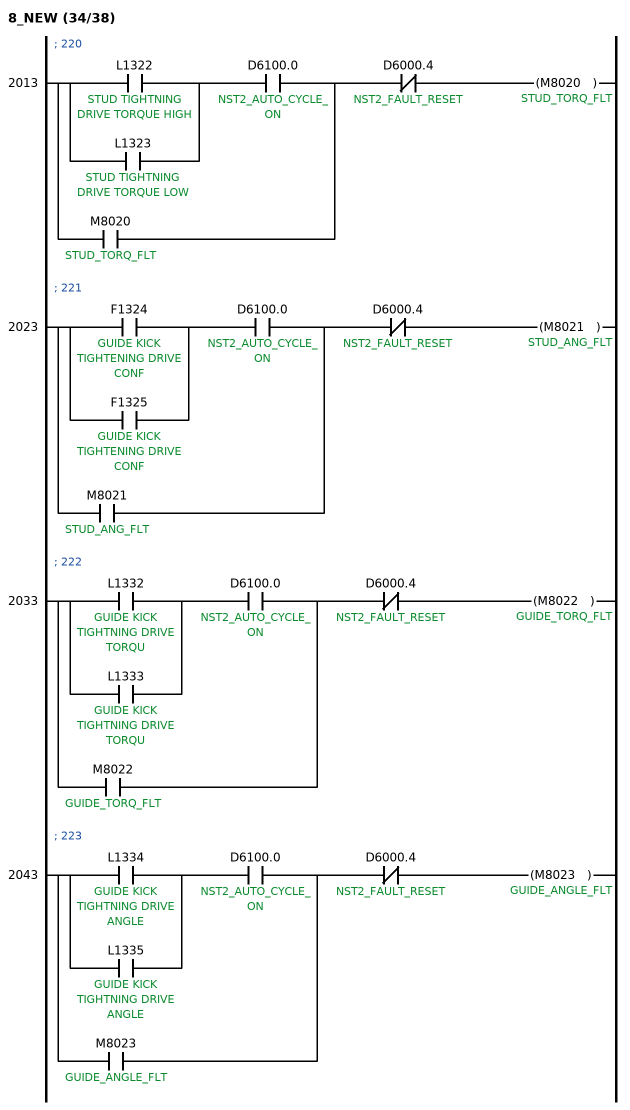
; 220
2013  LD      L1322  ; STUD TIGHTNING DRIVE TORQUE HIGH
      OR      L1323  ; STUD TIGHTNING DRIVE TORQUE LOW
      AND     D6100.0  ; NST2_AUTO_CYCLE_ON
      OR      M8020  ; STUD_TORQ_FLT
      ANI     D6000.4  ; NST2_FAULT_RESET
      OUT     M8020  ; STUD_TORQ_FLT
; 221
2023  LD      F1324  ; GUIDE KICK TIGHTENING DRIVE CONF
      OR      F1325  ; GUIDE KICK TIGHTENING DRIVE CONF
      AND     D6100.0  ; NST2_AUTO_CYCLE_ON
      OR      M8021  ; STUD_ANG_FLT
      ANI     D6000.4  ; NST2_FAULT_RESET
      OUT     M8021  ; STUD_ANG_FLT
; 222
2033  LD      L1332  ; GUIDE KICK TIGHTNING DRIVE TORQU
      OR      L1333  ; GUIDE KICK TIGHTNING DRIVE TORQU
      AND     D6100.0  ; NST2_AUTO_CYCLE_ON
      OR      M8022  ; GUIDE_TORQ_FLT
      ANI     D6000.4  ; NST2_FAULT_RESET
      OUT     M8022  ; GUIDE_TORQ_FLT
; 223
2043  LD      L1334  ; GUIDE KICK TIGHTNING DRIVE ANGLE
      OR      L1335  ; GUIDE KICK TIGHTNING DRIVE ANGLE
      AND     D6100.0  ; NST2_AUTO_CYCLE_ON
      OR      M8023  ; GUIDE_ANGLE_FLT
      ANI     D6000.4  ; NST2_FAULT_RESET
      OUT     M8023  ; GUIDE_ANGLE_FLT
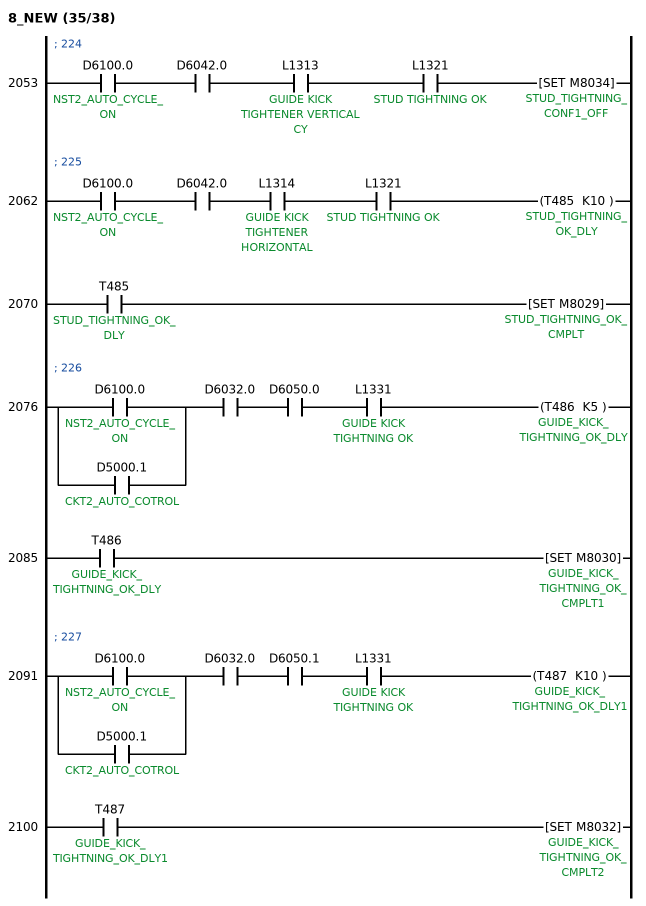
; 224
2053  LD      D6100.0  ; NST2_AUTO_CYCLE_ON
      AND     D6042.0
      AND     L1313  ; GUIDE KICK TIGHTENER VERTICAL CY
      AND     L1321  ; STUD TIGHTNING OK
      SET     M8034  ; STUD_TIGHTNING_CONF1_OFF
; 225
2062  LD      D6100.0  ; NST2_AUTO_CYCLE_ON
      AND     D6042.0
      AND     L1314  ; GUIDE KICK TIGHTENER HORIZONTAL
      AND     L1321  ; STUD TIGHTNING OK
      OUT     T485 K10  ; STUD_TIGHTNING_OK_DLY
2070  LD      T485  ; STUD_TIGHTNING_OK_DLY
      SET     M8029  ; STUD_TIGHTNING_OK_CMPLT
; 226
2076  LD      D6100.0  ; NST2_AUTO_CYCLE_ON
      OR      D5000.1  ; CKT2_AUTO_COTROL
      AND     D6032.0
      AND     D6050.0
      AND     L1331  ; GUIDE KICK TIGHTNING OK
      OUT     T486 K5  ; GUIDE_KICK_TIGHTNING_OK_DLY
2085  LD      T486  ; GUIDE_KICK_TIGHTNING_OK_DLY
      SET     M8030  ; GUIDE_KICK_TIGHTNING_OK_CMPLT1
; 227
2091  LD      D6100.0  ; NST2_AUTO_CYCLE_ON
      OR      D5000.1  ; CKT2_AUTO_COTROL
      AND     D6032.0
      AND     D6050.1
      AND     L1331  ; GUIDE KICK TIGHTNING OK
      OUT     T487 K10  ; GUIDE_KICK_TIGHTNING_OK_DLY1
2100  LD      T487  ; GUIDE_KICK_TIGHTNING_OK_DLY1
      SET     M8032  ; GUIDE_KICK_TIGHTNING_OK_CMPLT2
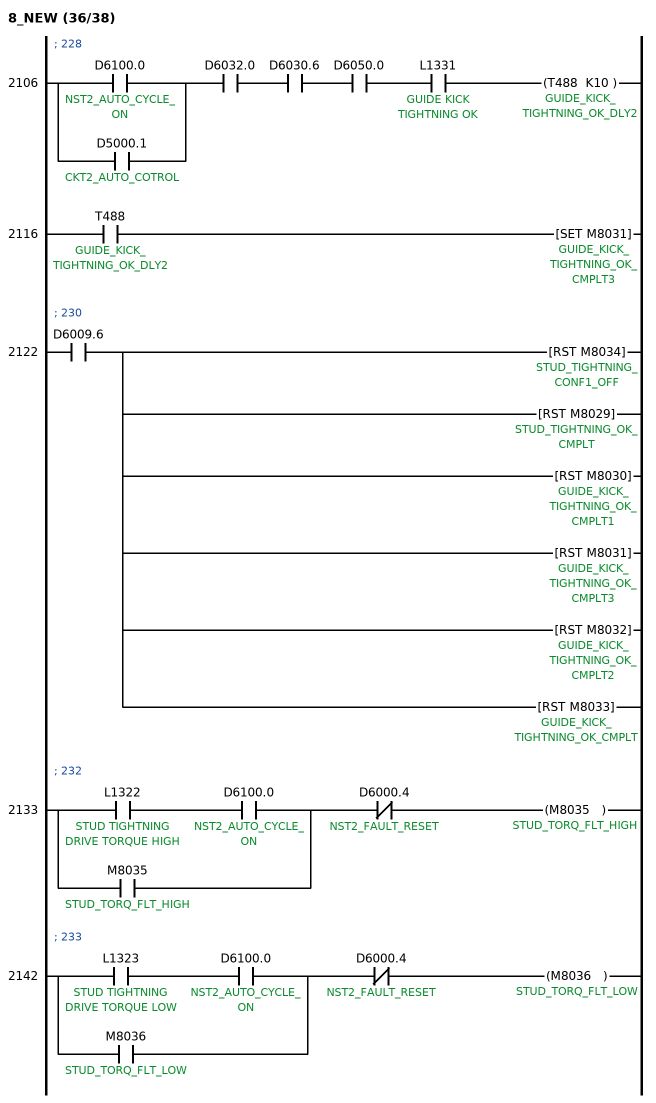
; 228
2106  LD      D6100.0  ; NST2_AUTO_CYCLE_ON
      OR      D5000.1  ; CKT2_AUTO_COTROL
      AND     D6032.0
      AND     D6030.6
      AND     D6050.0
      AND     L1331  ; GUIDE KICK TIGHTNING OK
      OUT     T488 K10  ; GUIDE_KICK_TIGHTNING_OK_DLY2
2116  LD      T488  ; GUIDE_KICK_TIGHTNING_OK_DLY2
      SET     M8031  ; GUIDE_KICK_TIGHTNING_OK_CMPLT3
; 230
2122  LD      D6009.6
      RST     M8034  ; STUD_TIGHTNING_CONF1_OFF
      RST     M8029  ; STUD_TIGHTNING_OK_CMPLT
      RST     M8030  ; GUIDE_KICK_TIGHTNING_OK_CMPLT1
      RST     M8031  ; GUIDE_KICK_TIGHTNING_OK_CMPLT3
      RST     M8032  ; GUIDE_KICK_TIGHTNING_OK_CMPLT2
      RST     M8033  ; GUIDE_KICK_TIGHTNING_OK_CMPLT
; 232
2133  LD      L1322  ; STUD TIGHTNING DRIVE TORQUE HIGH
      AND     D6100.0  ; NST2_AUTO_CYCLE_ON
      OR      M8035  ; STUD_TORQ_FLT_HIGH
      ANI     D6000.4  ; NST2_FAULT_RESET
      OUT     M8035  ; STUD_TORQ_FLT_HIGH
; 233
2142  LD      L1323  ; STUD TIGHTNING DRIVE TORQUE LOW
      AND     D6100.0  ; NST2_AUTO_CYCLE_ON
      OR      M8036  ; STUD_TORQ_FLT_LOW
      ANI     D6000.4  ; NST2_FAULT_RESET
      OUT     M8036  ; STUD_TORQ_FLT_LOW
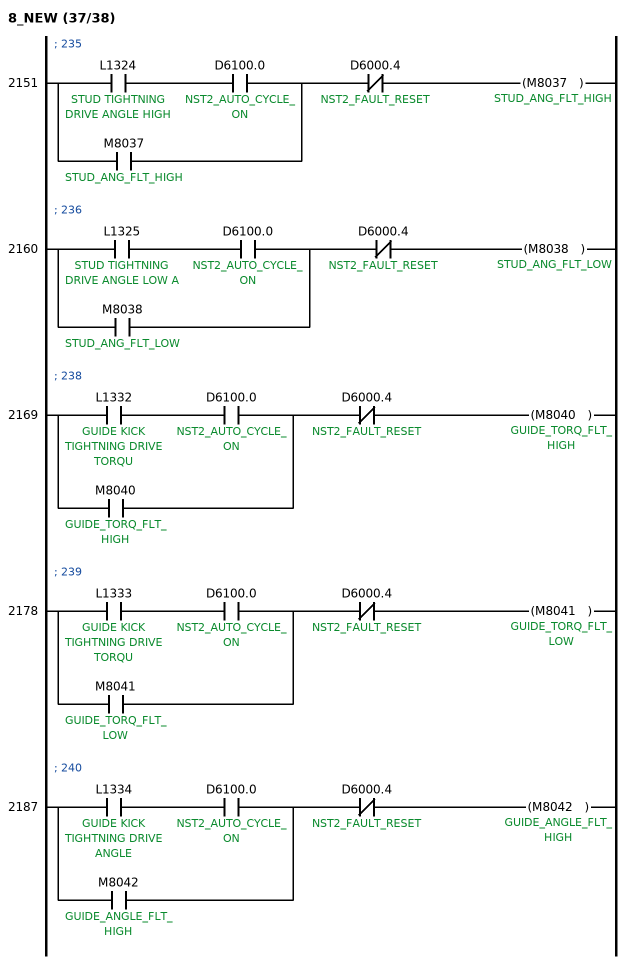
; 235
2151  LD      L1324  ; STUD TIGHTNING DRIVE ANGLE HIGH
      AND     D6100.0  ; NST2_AUTO_CYCLE_ON
      OR      M8037  ; STUD_ANG_FLT_HIGH
      ANI     D6000.4  ; NST2_FAULT_RESET
      OUT     M8037  ; STUD_ANG_FLT_HIGH
; 236
2160  LD      L1325  ; STUD TIGHTNING DRIVE ANGLE LOW A
      AND     D6100.0  ; NST2_AUTO_CYCLE_ON
      OR      M8038  ; STUD_ANG_FLT_LOW
      ANI     D6000.4  ; NST2_FAULT_RESET
      OUT     M8038  ; STUD_ANG_FLT_LOW
; 238
2169  LD      L1332  ; GUIDE KICK TIGHTNING DRIVE TORQU
      AND     D6100.0  ; NST2_AUTO_CYCLE_ON
      OR      M8040  ; GUIDE_TORQ_FLT_HIGH
      ANI     D6000.4  ; NST2_FAULT_RESET
      OUT     M8040  ; GUIDE_TORQ_FLT_HIGH
; 239
2178  LD      L1333  ; GUIDE KICK TIGHTNING DRIVE TORQU
      AND     D6100.0  ; NST2_AUTO_CYCLE_ON
      OR      M8041  ; GUIDE_TORQ_FLT_LOW
      ANI     D6000.4  ; NST2_FAULT_RESET
      OUT     M8041  ; GUIDE_TORQ_FLT_LOW
; 240
2187  LD      L1334  ; GUIDE KICK TIGHTNING DRIVE ANGLE
      AND     D6100.0  ; NST2_AUTO_CYCLE_ON
      OR      M8042  ; GUIDE_ANGLE_FLT_HIGH
      ANI     D6000.4  ; NST2_FAULT_RESET
      OUT     M8042  ; GUIDE_ANGLE_FLT_HIGH
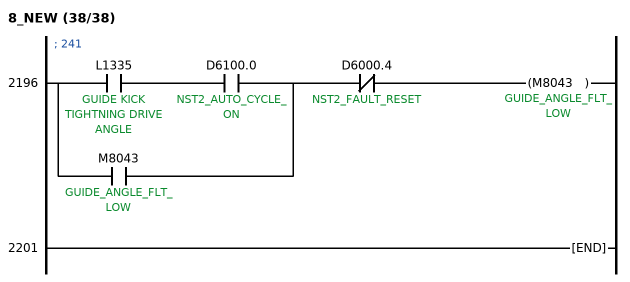
; 241
2196  LD      L1335  ; GUIDE KICK TIGHTNING DRIVE ANGLE
      AND     D6100.0  ; NST2_AUTO_CYCLE_ON
      OR      M8043  ; GUIDE_ANGLE_FLT_LOW
      ANI     D6000.4  ; NST2_FAULT_RESET
      OUT     M8043  ; GUIDE_ANGLE_FLT_LOW
2201  END
END_PROGRAM

PROGRAM 9_NEW  // ST3 CK2
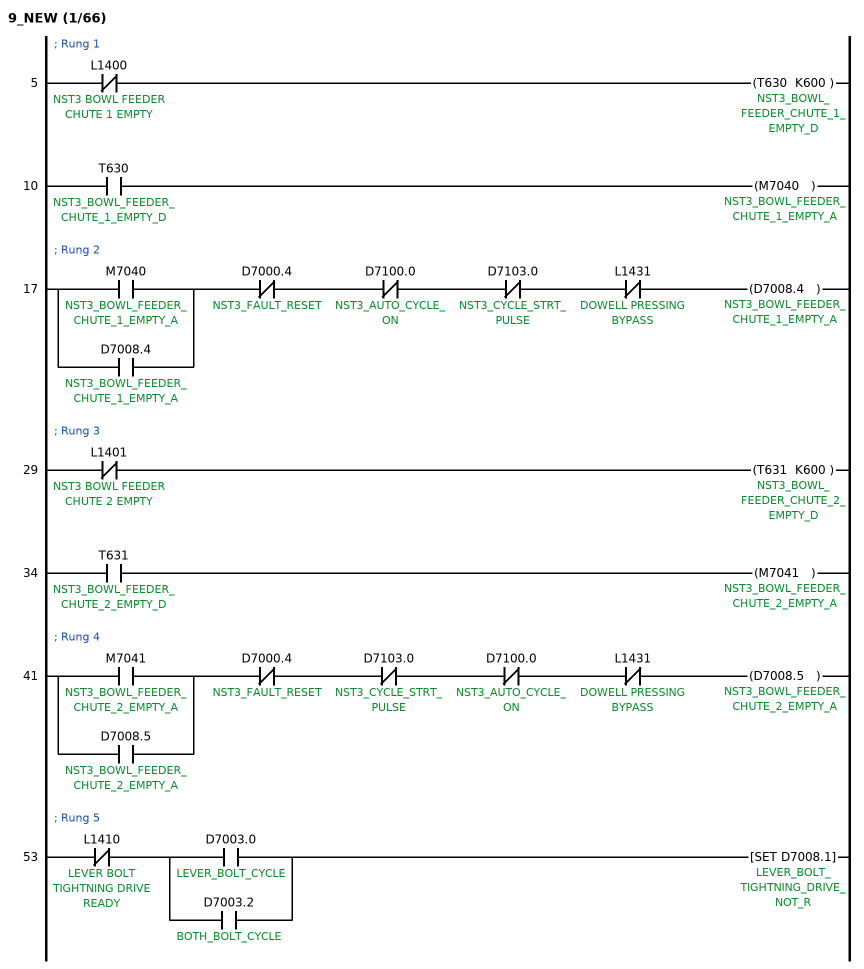
; Rung 1
5     LDI     L1400  ; NST3 BOWL FEEDER CHUTE 1 EMPTY
      OUT     T630 K600  ; NST3_BOWL_FEEDER_CHUTE_1_EMPTY_D
10    LD      T630  ; NST3_BOWL_FEEDER_CHUTE_1_EMPTY_D
      OUT     M7040  ; NST3_BOWL_FEEDER_CHUTE_1_EMPTY_A
; Rung 2
17    LD      M7040  ; NST3_BOWL_FEEDER_CHUTE_1_EMPTY_A
      OR      D7008.4  ; NST3_BOWL_FEEDER_CHUTE_1_EMPTY_A
      ANI     D7000.4  ; NST3_FAULT_RESET
      ANI     D7100.0  ; NST3_AUTO_CYCLE_ON
      ANI     D7103.0  ; NST3_CYCLE_STRT_PULSE
      ANI     L1431  ; DOWELL PRESSING BYPASS
      OUT     D7008.4  ; NST3_BOWL_FEEDER_CHUTE_1_EMPTY_A
; Rung 3
29    LDI     L1401  ; NST3 BOWL FEEDER CHUTE 2 EMPTY
      OUT     T631 K600  ; NST3_BOWL_FEEDER_CHUTE_2_EMPTY_D
34    LD      T631  ; NST3_BOWL_FEEDER_CHUTE_2_EMPTY_D
      OUT     M7041  ; NST3_BOWL_FEEDER_CHUTE_2_EMPTY_A
; Rung 4
41    LD      M7041  ; NST3_BOWL_FEEDER_CHUTE_2_EMPTY_A
      OR      D7008.5  ; NST3_BOWL_FEEDER_CHUTE_2_EMPTY_A
      ANI     D7000.4  ; NST3_FAULT_RESET
      ANI     D7103.0  ; NST3_CYCLE_STRT_PULSE
      ANI     D7100.0  ; NST3_AUTO_CYCLE_ON
      ANI     L1431  ; DOWELL PRESSING BYPASS
      OUT     D7008.5  ; NST3_BOWL_FEEDER_CHUTE_2_EMPTY_A
; Rung 5
53    LDI     L1410  ; LEVER BOLT TIGHTNING DRIVE READY
      LD      D7003.0  ; LEVER_BOLT_CYCLE
      OR      D7003.2  ; BOTH_BOLT_CYCLE
      ANB
      SET     D7008.1  ; LEVER_BOLT_TIGHTNING_DRIVE_NOT_R
